// TIA Portal project "MyOpennessGeneratedProject" (V16)

(* hardware
DEVICE "S71500/ET200MP-Station_1"  S7-1500 station
   slot 0: "Profilschiene_0"  Rack  6ES7 590-1***0-0AA0
   slot 1: "PLC_1"  CPU 1513F-1 PN  6ES7 513-1FL01-0AB0  V2.0
      slot 3: "CPU-Display_1"  6ES7591-1AA00-0AA0
   slot 2: "DI 32x24VDC HF_1"  DI 32x24VDC HF  6ES7 521-1BL00-0AB0  V1.0
   slot 3: "DQ 32x24VDC/0.5A ST_1"  DQ 32x24VDC/0.5A ST  6ES7 522-1BL00-0AB0  V1.0
   slot 4: "AI 8xU/I/RTD/TC ST_1"  AI 8xU/I/RTD/TC ST  6ES7 531-7KF00-0AB0  V1.0
DEVICE "ET 200SP-Station_1"  ET 200SP-Station
   slot 0: "Baugruppenträger_0"  Rack  6ES5 710-8MAx1
   slot 0: "ET200SP"  IM 155-6 PN ST  6ES7 155-6AU00-0BN0  V1.0
   slot 1: "DI 8x24VDC ST_1"  DI 8x24VDC ST  6ES7 131-6BF00-0BA0  V1.0
      slot 1: "DI 8x24VDC ST_1"  DI 8x24VDC ST
   slot 2: "DI 8x24VDC ST_2"  DI 8x24VDC ST  6ES7 131-6BF00-0BA0  V1.0
      slot 1: "DI 8x24VDC ST_2"  DI 8x24VDC ST
   slot 3: "DQ 16x24VDC/0.5A ST_1"  DQ 16x24VDC/0.5A ST  6ES7 132-6BH00-0BA0  V1.0
      slot 1: "DQ 16x24VDC/0.5A ST_1"  DQ 16x24VDC/0.5A ST
   slot 4: "AI 4xU/I 2-wire ST_1"  AI 4xU/I 2-wire ST  6ES7 134-6HD00-0BA1  V1.0
      slot 1: "AI 4xU/I 2-wire ST_1"  AI 4xU/I 2-wire ST
   slot 5: "AQ 4xU/I ST_1"  AQ 4xU/I ST  6ES7 135-6HD00-0BA1  V1.0
      slot 1: "AQ 4xU/I ST_1"  AQ 4xU/I ST
   slot 6: "Servermodul_1"  Server module  6ES7 193-6PA00-0AA0  V1.1
      slot 1: "Servermodul_1"  Server module
   slot 127: "BA 2xRJ45"  BA 2xRJ45  6ES7 193-6AR00-0AA0  V0.0
      slot 1: "Port_1"  X1 P1 R  6ES7 193-6AR00-0AA0  V0.0
      slot 2: "Port_2"  X1 P2 R  6ES7 193-6AR00-0AA0  V0.0
DEVICE "Touchpanel"  TP700 Comfort
   slot 0: "Touchpanel"  TP700 Comfort  6AV2 124-0GC01-0AX0  16.0.0.0
   slot 1: "HMI_RT_1"  TP700 Comfort  6AV2 124-0GC01-0AX0  16.0.0.0
   slot 5: "Touchpanel"  PROFINET Interface  IE_CP  16.0.0.0
      slot 1: "PROFINET Interface_1"  PROFINET Interface
         slot 1: "PORT_2"  Port  1.0.0.0
         slot 2: "PORT_1"  Port  1.0.0.0
   slot 7: "Touchpanel.MPI/DP_CP"  MPI/DP Interface  MPI-DP_CP  16.0.0.0
*)

// ===== PLC "PLC_1"  CPU 1513F-1 PN =====
// protected blocks, not shown: "FC_Signal"

VAR_GLOBAL   // PLC tag table "My_Tags"
   "S_Fault3" AT %E0.6 : Bool;   // Schalter Störung 3 / S_Fault3
   "M_JogRight" AT %M16.2 : Bool;   // Merker Tippen Rechts / Memory bit Jog conveyor RIGHT
   "M_AutoRight" AT %M16.4 : Bool;   // Merker Auto Rechts / Memory bit Conveyor AUTO RIGHT
   "M_ConvFault" AT %M17.0 : Bool;   // Merker Bandlauf-Störung / Memory bit Conveyor fault
   "S_Acknowledge" AT %E0.7 : Bool;   // Taster Quittierung / S_Acknowledge
   "P_Operation" AT %A0.1 : Bool;   // Meldeleuchte Betrieb EIN / Indicator light Operation ON
   "P_Fault" AT %A0.7 : Bool;   // Anzeige Band-Störung / Indicator light for fault
   "M_AuxFault1" AT %M17.1 : Bool;   // Edge auxiliary memory bit Fault 1 / Flanken-Hilfsmerker Störung 1
   "P_Fault1" AT %A0.2 : Bool;   // Anzeige Störung 1 / Indicator light for fault1
   "P_Fault2" AT %A0.3 : Bool;   // Anzeige Störung 2 / Indicator light for fault2
   "S_Fault1" AT %E0.4 : Bool;   // Schalter Störung 1 / S_Fault1
   "S_Fault2" AT %E0.5 : Bool;   // Schalter Störung 2 / S_Fault2
   "P_Fault3" AT %A0.4 : Bool;   // Anzeige Störung 3 / Indicator light for fault3
   "M_AuxOpON" AT %M15.1 : Bool;   // Edge auxiliary memory bit Operation ON / Flanken-Hilfsmerker Anlage EIN
   "M_ActSetp" AT %M18.4 : Bool;   // Merker Ist-Stückzahl=Soll-Stückzah / Memory bit Actual- has reached Setpoint number
   "S_OperationON" AT %E0.1 : Bool;   // Taster Betrieb EIN / S_OperationON
   "S_OperationOFF" AT %E0.0 : Bool;   // Taster Betrieb AUS / S_OperationOFF
   "S_Right" AT %E0.2 : Bool;   // Taster Tippen Rechts / S_Right
   "S_Left" AT %E0.3 : Bool;   // Taster Tippen Links / S_Left
   "M_StorFault1" AT %M17.2 : Bool;   // Memory bit for storing Fault 1 / Merker Meldespeicher Störung 1
   "M_AuxFault2" AT %M17.3 : Bool;   // Edge auxiliary memory bit Fault 2 / Flanken-Hilfsmerker Störung 2
   "M_StorFault2" AT %M17.4 : Bool;   // Memory bit for storing Fault 2 / Merker Meldespeicher Störung 2
   "M_AuxLB" AT %M16.0 : Bool;   // Edge auxiliary memory bit Light barrier / Flanken-Hilfsmerker Lichtschranke
END_VAR

VAR_GLOBAL   // PLC tag table "Var_Clocks"
   "Clock_Byte" AT %MB10 : Byte;
   "Clock_10Hz" AT %M10.0 : Bool;
   "Clock_5Hz" AT %M10.1 : Bool;
   "Clock_2.5Hz" AT %M10.2 : Bool;
   "Clock_2Hz" AT %M10.3 : Bool;
   "Clock_1.25Hz" AT %M10.4 : Bool;
   "Clock_1Hz" AT %M10.5 : Bool;
   "Clock_0.625Hz" AT %M10.6 : Bool;
   "Clock_0.5Hz" AT %M10.7 : Bool;
END_VAR

VAR_GLOBAL   // PLC tag table "Conveyor"
   "B_LB" AT %I20.0 : Bool;   // Lichtschranke / Light barrier
   "S_Bay1" AT %I20.1 : Bool;   // Taster Platz 1 / Momentary contact Bay 1
   "S_Bay2" AT %I20.2 : Bool;   // Taster Platz 2 / Momentary contact Bay 2
   "S_Bay3" AT %I20.3 : Bool;   // Taster Platz 3 / Momentary contact Bay 3
   "S_BayLB" AT %I20.4 : Bool;   // Taster Lichtschranken-Platz / Momentary contact Light barrier bay
   "B_Bay1" AT %I20.5 : Bool;   // Initiator Platz 1 / Proximity sensor Bay 1
   "B_Bay2" AT %I20.6 : Bool;   // Initiator Platz 2 / Proximity sensor Bay 2
   "B_Bay3" AT %I20.7 : Bool;   // Initiator Platz 3 / Proximity sensor Bay 3
   "P_Bay1" AT %Q4.1 : Bool;   // Meldeleuchte Platz 1 / Indicator light Bay 1
   "P_Bay2" AT %Q4.2 : Bool;   // Meldeleuchte Platz 2 / Indicator light Bay 2
   "P_Bay3" AT %Q4.3 : Bool;   // Meldeleuchte Platz 3 / Indicator light Bay 3
   "P_BayLB" AT %Q4.4 : Bool;   // Meldeleuchte Lichtschranken-Platz / Indicator light Light barrier bay
   "K_Right" AT %Q4.5 : Bool;   // Bandmotor Rechts / Run conveyor RIGHT
   "K_Left" AT %Q4.6 : Bool;   // Bandmotor Links / Run conveyor LEFT
   "P_Horn" AT %Q4.7 : Bool;   // Hupe / Horn
END_VAR

DATA_BLOCK "iDB_FB_Mode"   // DB1
{ S7_Optimized_Access := 'TRUE' }
VERSION : 0.1
// stored: InstanceOfName FB_Mode
"FB_Mode"
BEGIN
END_DATA_BLOCK

DATA_BLOCK "DB_OP"   // DB2
{ S7_Optimized_Access := 'TRUE' }
VERSION : 0.1
   VAR
      AcknFault : Bool;
      JogLeft : Bool;
      JogRight : Bool;
      OperationOFF : Bool;
      OperationON : Bool;
   END_VAR
BEGIN
END_DATA_BLOCK

FUNCTION_BLOCK "FB_Mode"   // FB1, FBD
{ S7_Optimized_Access := 'TRUE' }
VERSION : 0.1
   VAR_INPUT
      OperationON : Bool;
      OperationOff : Bool;
   END_VAR
   VAR_IN_OUT
      Operation_State : Bool;
   END_VAR
   VAR
      M_AuxOpON : Bool;
   END_VAR
   VAR_TEMP   // added for the SCL form of the ladder/FBD networks
      _w1 : Bool;
   END_VAR
BEGIN

REGION Network 1: Betriebsartenwahl
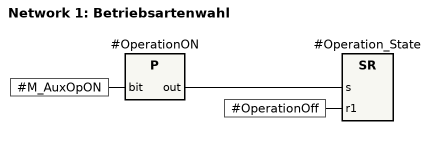
   #_w1 := #OperationON AND NOT #M_AuxOpON;   // rising edge of #OperationON
   #M_AuxOpON := #OperationON;
   IF #_w1 THEN
       #Operation_State := TRUE;   // SR flip-flop
   END_IF;
   IF #OperationOff THEN #Operation_State := FALSE; END_IF;
END_REGION
END_FUNCTION_BLOCK

FUNCTION "FC_Conveyor" : Void   // FC16, FBD
{ S7_Optimized_Access := 'TRUE' }
VERSION : 0.1
   VAR_INPUT
      RequestRight : Bool;
      Request_Left : Bool;
      OperationState : Bool;
      Bay1_Occupied : Bool;
      Bay2_Occupied : Bool;
      RequestBay1 : Bool;
      RequestBay2 : Bool;
      LBNotOccupied : Bool;
   END_VAR
   VAR_OUTPUT
      GoRight : Bool;
      GoLeft : Bool;
   END_VAR
   VAR_IN_OUT
      MemForAutoRight : Bool;
      MemForManRight : Bool;
   END_VAR
BEGIN

REGION Network 1: Hand Rechts
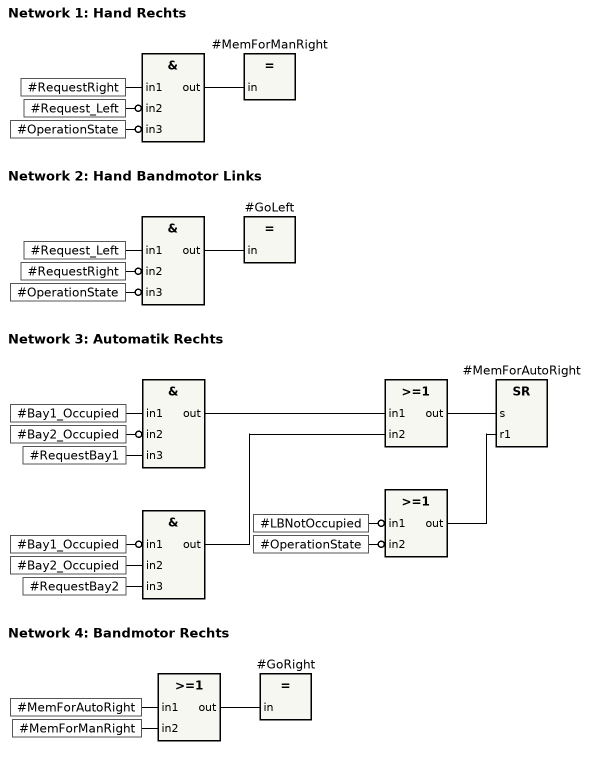
   #MemForManRight := #RequestRight AND NOT #Request_Left AND NOT #OperationState;
END_REGION

REGION Network 2: Hand Bandmotor Links
   #GoLeft := #Request_Left AND NOT #RequestRight AND NOT #OperationState;
END_REGION

REGION Network 3: Automatik Rechts
   IF (#Bay1_Occupied AND NOT #Bay2_Occupied AND #RequestBay1) OR (NOT #Bay1_Occupied AND #Bay2_Occupied AND #RequestBay2) THEN
       #MemForAutoRight := TRUE;   // SR flip-flop
   END_IF;
   IF NOT #LBNotOccupied OR NOT #OperationState THEN #MemForAutoRight := FALSE; END_IF;
END_REGION

REGION Network 4: Bandmotor Rechts
   #GoRight := #MemForAutoRight OR #MemForManRight;
END_REGION
END_FUNCTION

ORGANIZATION_BLOCK "Main"   // OB1, FBD, ProgramCycle
TITLE = "Main Program Sweep (Cycle)"
{ S7_Optimized_Access := 'TRUE' }
VERSION : 0.1
   VAR_INPUT
      Initial_Call : Bool;   // Initial call of this OB
      Remanence : Bool;   // =True, if remanent data are available
   END_VAR
BEGIN

REGION Network 1
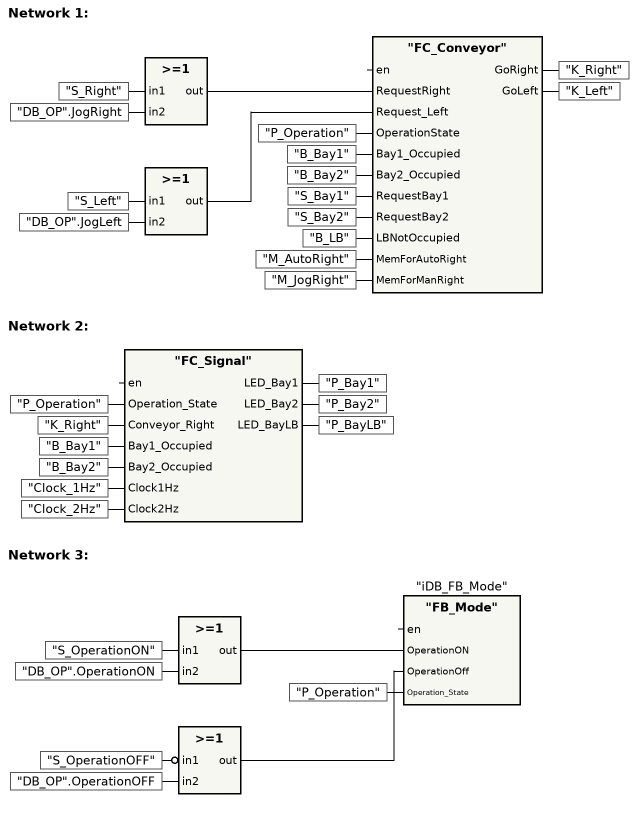
   "FC_Conveyor"(RequestRight := "S_Right" OR "DB_OP".JogRight,
                 Request_Left := "S_Left" OR "DB_OP".JogLeft,
                 OperationState := "P_Operation",
                 Bay1_Occupied := "B_Bay1",
                 Bay2_Occupied := "B_Bay2",
                 RequestBay1 := "S_Bay1",
                 RequestBay2 := "S_Bay2",
                 LBNotOccupied := "B_LB",
                 MemForAutoRight := "M_AutoRight",
                 MemForManRight := "M_JogRight",
                 GoRight => "K_Right",
                 GoLeft => "K_Left");
END_REGION

REGION Network 2
   "FC_Signal"(Operation_State := "P_Operation",
               Conveyor_Right := "K_Right",
               Bay1_Occupied := "B_Bay1",
               Bay2_Occupied := "B_Bay2",
               Clock1Hz := "Clock_1Hz",
               Clock2Hz := "Clock_2Hz",
               LED_Bay1 => "P_Bay1",
               LED_Bay2 => "P_Bay2",
               LED_BayLB => "P_BayLB");
END_REGION

REGION Network 3
   "iDB_FB_Mode"(OperationON := "S_OperationON" OR "DB_OP".OperationON,   // "FB_Mode"
                 OperationOff := NOT "S_OperationOFF" OR "DB_OP".OperationOFF,
                 Operation_State := "P_Operation");
END_REGION
END_ORGANIZATION_BLOCK

// ===== PLC "S7-1500"   =====

(* ===== HMI "HMI_RT_1" =====
system functions are stored by id; their names below are inferred from use
connection "HMI_Verbindung_2": ETHERNET, S7_1500_OMS

HMI tags "Standard-Variablentabelle"
   "P_Operation" : Bool = PLC P_Operation AT %Q0.1, 100 ms   // Meldeleuchte Betrieb EIN / Signalling light Plant ON
   "P_BayLB" : Bool = PLC P_BayLB AT %Q4.4, 100 ms   // Meldeleuchte Platz LS / Indicator light Bay LB
   "P_Bay1" : Bool = PLC P_Bay1 AT %Q4.1, 100 ms   // Meldeleuchte Platz 1 / Indicator light Bay 1
   "P_Bay2" : Bool = PLC P_Bay2 AT %Q4.2, 100 ms   // Meldeleuchte Platz 2 / Indicator light Bay 2
   "B_Bay1" : Bool = PLC B_Bay1 AT %I20.5, 100 ms   // Initiator Platz 1 / Indicator light Bay 1
   "B_Bay2" : Bool = PLC B_Bay2 AT %I20.6, 100 ms   // Initiator Platz 2 / Indicator light Bay 2
   "B_LB" : Bool = PLC B_LB AT %I20.0, 100 ms   // Lichtschranke / Light barrier
   "M_ConvFault" : Bool = PLC M_ConvFault AT %M17.0, 100 ms   // Merker Bandlauf-Störung / Memory bit Conveyor fault
   "DB_OP_OperationOFF" : Bool = PLC DB_OP.OperationOFF, 100 ms   // Anlage AUS / Operation OFF
   "DB_OP_OperationON" : Bool = PLC DB_OP.OperationON, 100 ms   // Anlage EIN / Operation ON
   "DB_OP_JogLeft" : Bool = PLC DB_OP.JogLeft, 100 ms   // Bandmotor Tippen LINKS (Touchpanel) / Jog conveyor motor Left (Touchpanel)
   "DB_OP_AcknFault" : Bool = PLC DB_OP.AcknFault, 100 ms   // Band-Störung quittieren (Touchpanel) / Acknowledge conveyor fault (Touchpanel)
   "DB_OP_JogRight" : Bool = PLC DB_OP.JogRight, 100 ms   // Bandmotor Tippen RECHTS (Touchpanel) / Jog conveyor motor Right (Touchpanel)
   "P_Bay3" : Bool = PLC P_Bay3 AT %Q4.3, 100 ms   // Meldeleuchte Platz 3 / Indicator light Bay 3
   "B_Bay3" : Bool = PLC B_Bay3 AT %I20.7, 100 ms   // Initiator Patz 3 / Indicator light Bay 3
   "ScreenNr" : Int, internal

text list "Betrieb": 0 'Betrieb AUS / Plant OFF'; 1 'Betrieb EIN / Plant ON'

screen "Bild_1" 800x446
   Button "Schaltfläche_1" at 6,392 size 786x48; TextOn 'Conveyor_1'; TextOff 'Go to Conveyor screen / Go to conveyor'
      on Click: ActivateScreenByNumber("ScreenNr", 0)
   TextField "Textfeld_1" at 56,25 size 744x29; Text 'Welcome to the Openness-Generated Screens of this HMI! / Welcome to the Openness Generated Screens of this Touchpanel!'
   GraphicView "Grafikanzeige_1" at 316,142 size 227x96; Picture "Grafik_2"

screen "Conveyor_1" 800x446
   GraphicView "Grafikanzeige_1" at 140,164 size 520x160; Picture "Grafik_1"
   Button "Schaltfläche_1" at 10,6 size 121x68; TextOff 'Betrieb EIN Plant ON'
      on Release: ResetBit("DB_OP_OperationON")
      on Press: SetBit("DB_OP_OperationON")
   Button "Schaltfläche_2" at 669,6 size 120x68; TextOff 'Betrieb AUS Plant OFF'
      on Release: ResetBit("DB_OP_OperationOFF")
      on Press: SetBit("DB_OP_OperationOFF")
   Button "Schaltfläche_3" at 10,372 size 121x68; TextOff 'Fehler Quittierung Error acknowledge'
      on Release: ResetBit("DB_OP_AcknFault")
      on Press: SetBit("DB_OP_AcknFault")
   Button "Schaltfläche_5" at 669,196 size 120x68; TextOff 'Tippen Rechts Jog right'
      on Release: ResetBit("DB_OP_JogRight")
      on Press: SetBit("DB_OP_JogRight")
   Button "Schaltfläche_6" at 10,196 size 121x68; TextOff 'Tippen Links Jog left'
      on Release: ResetBit("DB_OP_JogLeft")
      on Press: SetBit("DB_OP_JogLeft")
   Circle "Kreis_5" at 275,272 size 12x12
      Visibility <- "P_Bay1"
   Circle "Kreis_6" at 347,272 size 12x12
      Visibility <- "P_Bay2"
   Circle "Kreis_7" at 418,272 size 12x12
      Visibility <- "P_Bay3"
   Circle "Kreis_8" at 568,272 size 12x12
      Visibility <- "P_BayLB"
   TextField "Textfeld_3" at 246,318 size 318x34; Text 'Bandlauf-Störung / Conveyor Fault'
      Visibility <- "M_ConvFault"
   SymbolicIOField "Symbolisches EA-Feld_1" at 184,21 size 438x38; TextOn '1'; TextOff '0'; TextList "Betrieb"
      ProcessValue <- "P_Operation"
   Rectangle "Rechteck_1" at 533,183 size 14x13
      Visibility <- "B_LB"
   Rectangle "Rechteck_2" at 452,182 size 13x12
      Visibility <- "B_Bay3"
   Rectangle "Rechteck_3" at 380,182 size 13x12
      Visibility <- "B_Bay2"
   Rectangle "Rechteck_4" at 308,182 size 13x12
      Visibility <- "B_Bay1"
   Button "OBJECT_4" at 667,372 size 125x68; TextOff 'Stop RT / Exit RT'
      on Release: StopRuntime(0)
*)

(* ===== HMI "HMI_RT_1" =====
system functions are stored by id; their names below are inferred from use

text list "Betrieb": 0 'Betrieb AUS / Plant OFF'; 1 'Betrieb EIN / Plant ON'

screen "hg1jahs3gd0jgsa09837c03-996a-4fc1-9506-5bab3cd600520" 800x446
   GraphicView "Grafikanzeige_1" at 140,164 size 520x160; Picture "Grafik_1"
   Button "Schaltfläche_1" at 10,6 size 121x68; TextOff 'Betrieb EIN Plant ON'
      on Release: ResetBit("DB_OP_OperationON")
      on Press: SetBit("DB_OP_OperationON")
   Button "Schaltfläche_2" at 669,6 size 120x68; TextOff 'Betrieb AUS Plant OFF'
      on Release: ResetBit("DB_OP_OperationOFF")
      on Press: SetBit("DB_OP_OperationOFF")
   Button "Schaltfläche_3" at 10,372 size 121x68; TextOff 'Fehler Quittierung Error acknowledge'
      on Release: ResetBit("DB_OP_AcknFault")
      on Press: SetBit("DB_OP_AcknFault")
   Button "Schaltfläche_5" at 669,196 size 120x68; TextOff 'Tippen Rechts Jog right'
      on Release: ResetBit("DB_OP_JogRight")
      on Press: SetBit("DB_OP_JogRight")
   Button "Schaltfläche_6" at 10,196 size 121x68; TextOff 'Tippen Links Jog left'
      on Release: ResetBit("DB_OP_JogLeft")
      on Press: SetBit("DB_OP_JogLeft")
   Circle "Kreis_5" at 275,272 size 12x12
      Visibility <- "P_Bay1"
   Circle "Kreis_6" at 347,272 size 12x12
      Visibility <- "P_Bay2"
   Circle "Kreis_7" at 418,272 size 12x12
      Visibility <- "P_Bay3"
   Circle "Kreis_8" at 568,272 size 12x12
      Visibility <- "P_BayLB"
   TextField "Textfeld_3" at 246,318 size 318x34; Text 'Bandlauf-Störung / Conveyor Fault'
      Visibility <- "M_ConvFault"
   SymbolicIOField "Symbolisches EA-Feld_1" at 184,21 size 438x38; TextOn '1'; TextOff '0'; TextList "Betrieb"
      ProcessValue <- "P_Operation"
   Rectangle "Rechteck_1" at 533,183 size 14x13
      Visibility <- "B_LB"
   Rectangle "Rechteck_2" at 452,182 size 13x12
      Visibility <- "B_Bay3"
   Rectangle "Rechteck_3" at 380,182 size 13x12
      Visibility <- "B_Bay2"
   Rectangle "Rechteck_4" at 308,182 size 13x12
      Visibility <- "B_Bay1"
   Button "OBJECT_4" at 667,372 size 125x68; TextOff 'Stop RT / Exit RT'
      on Release: StopRuntime(0)
*)